FUNCTION_BLOCK L2_ASetupREQHDLR (* Basic Function Block Type *)
  (* Standard: 61499-2 *)
  (* Version 0.0, 2014-11-28, EQUEROL, UJI *)
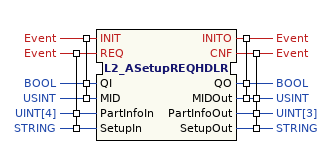
  EVENT_INPUT
    INIT WITH MID, QI; (* Initialization Request *)
    REQ WITH PartInfoIn, SetupIn; (* Normal Execution Request *)
  END_EVENT
  EVENT_OUTPUT
    INITO WITH QO, MIDOut; (* Initialization Confirm *)
    CNF WITH PartInfoOut, MIDOut, SetupOut; (* Execution Confirmation *)
  END_EVENT
  VAR_INPUT
    QI : BOOL;
    MID : USINT; (* Machine identifier *)
    PartInfoIn : ARRAY [0..3] OF UINT; (* Part ID, family, type, MID *)
    SetupIn : STRING; (* Subphase to execute *)
  END_VAR
  VAR_OUTPUT
    QO : BOOL;
    MIDOut : USINT; (* Machine identifier *)
    PartInfoOut : ARRAY [0..2] OF UINT; (* Part identifier, family and type *)
    SetupOut : STRING; (* Subphase to execute *)
  END_VAR
  VAR
    Accepted : BOOL := FALSE; (* This variable allow to diferentiate between accepted and rejected request *)
    i : USINT := 0; (* loop variable *)
  END_VAR
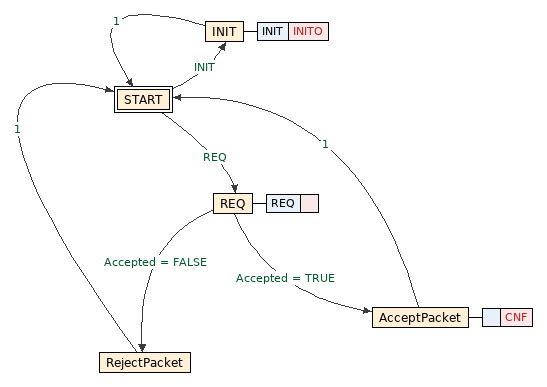
  EC_STATES
    START; (* Initial State *)
    INIT : INIT -> INITO; (* Initialization *)
    REQ : REQ; (* Normal execution *)
    AcceptPacket : -> CNF;
    RejectPacket;
  END_STATES
  EC_TRANSITIONS
    START TO INIT := INIT;
    INIT TO START := 1;
    START TO REQ := REQ;
    REQ TO AcceptPacket := Accepted = TRUE;
    REQ TO RejectPacket := Accepted = FALSE;
    RejectPacket TO START := 1;
    AcceptPacket TO START := 1;
  END_TRANSITIONS
  ALGORITHM INIT IN ST: (* Initialization algorithm *)
QO := QI;
MIDOut := MID;
  END_ALGORITHM
  ALGORITHM REQ IN ST: (* Normally executed algorithm *)
IF PartInfoIn[3] = MID THEN
	(*The received packet is for this machine, map outputs*)
	Accepted := TRUE;
	PartInfoOut[0] := PartInfoIn[0];
	PartInfoOut[1] := PartInfoIn[1];
	PartInfoOut[2] := PartInfoIn[2];
	PartInfoOut[3] := PartInfoIn[3];
	SetupOut :=SetupIn;
ELSE
	Accepted := FALSE;
END_IF;
  END_ALGORITHM
END_FUNCTION_BLOCK
